FUNCTION_BLOCK FB_Object IMPLEMENTS I_Object
VAR_INPUT
END_VAR
VAR_OUTPUT
END_VAR
VAR
	_ipObject 			: I_Object := 0;
END_VAR

METHOD Destruct : BOOL
// object destructor
IF (_ipObject <> 0) THEN
	_ipObject.Destruct();
	_ipObject := 16#0;
END_IF
END_METHOD

PROPERTY ipObject : I_Object
GET
ipObject := this^._ipObject;
END_GET
SET
IF (ipObject<>0) THEN
	THIS^._ipObject := ipObject;
ELSE
	THIS^._ipObject := 0;
END_IF
END_SET
END_PROPERTY

METHOD M_GetObjectDescription : STRING
M_GetObjectDescription := 'Error';
IF (_ipObject <> 0) THEN
	M_GetObjectDescription := _ipObject.M_GetObjectDescription();
END_IF
END_METHOD

{warning 'add method implementation'}
METHOD M_Reset : BOOL
END_METHOD

{warning 'add method implementation'}
METHOD M_Start : BOOL
END_METHOD

{warning 'add property implementation'}
PROPERTY P_Status : DWORD
GET
END_GET
END_PROPERTY

END_FUNCTION_BLOCK

(* stored: Version 1.1.0.1, ProductVersion 3.1.4024.12
   POU FB_Object: Id {630e43f6-dabf-46f7-9bf3-2d4a36c97869}, SpecialFunc None
   Method Destruct: Id {de441e1b-6ff0-4559-b14e-30118cac3714}
   Property ipObject: Id {168e2159-3eaa-4ebc-a520-7638afede6c1}
   Get Get: Id {f85965ae-377d-47df-896d-df9934ec4ce9}
   Set Set: Id {1b05c7f8-147d-4f4a-8f9a-9b12fef8b868}
   Method M_GetObjectDescription: Id {e6aa9a81-1045-4f48-bbfe-5b0657fccc0b}
   Method M_Reset: Id {69f84b58-a728-441f-89f7-b0d4aaefd84f}
   Method M_Start: Id {3101429e-36b4-41b5-8a3c-8f509a015f33}
   Property P_Status: Id {0a05751c-5b08-4f3e-8cc2-7eb12d7f6de2}
   Get Get: Id {a37098e4-8122-444e-a5d2-398549f50b43} *)
